// Mitsubishi GX Works2 project: 41715072   PLC: Q00J

PROGRAM MAIN
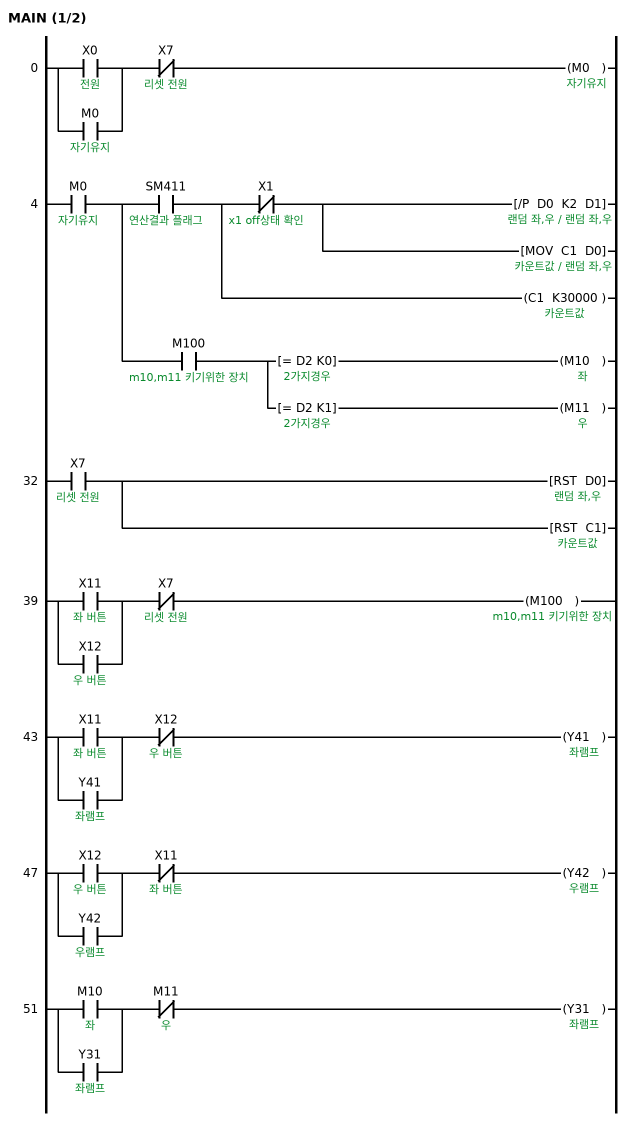
0     LD      X0  ; 전원
      OR      M0  ; 자기유지
      ANI     X7  ; 리셋 전원
      OUT     M0  ; 자기유지
4     LD      M0  ; 자기유지
      MPS
      AND     SM411  ; 연산결과 플래그
      MPS
      ANI     X1  ; x1 off상태 확인
      /P      D0 K2 D1  ; 랜덤 좌,우 / 랜덤 좌,우
      MOV     C1 D0  ; 카운트값
      MPP
      OUT     C1 K30000  ; 카운트값
      MPP
      AND     M100  ; m10,m11 키기위한 장치
      MPS
      AND=    D2 K0  ; 2가지경우
      OUT     M10  ; 좌
      MPP
      AND=    D2 K1  ; 2가지경우
      OUT     M11  ; 우
32    LD      X7  ; 리셋 전원
      RST     D0  ; 랜덤 좌,우
      RST     C1  ; 카운트값
39    LD      X11  ; 좌 버튼
      OR      X12  ; 우 버튼
      ANI     X7  ; 리셋 전원
      OUT     M100  ; m10,m11 키기위한 장치
43    LD      X11  ; 좌 버튼
      OR      Y41  ; 좌램프
      ANI     X12  ; 우 버튼
      OUT     Y41  ; 좌램프
47    LD      X12  ; 우 버튼
      OR      Y42  ; 우램프
      ANI     X11  ; 좌 버튼
      OUT     Y42  ; 우램프
51    LD      M10  ; 좌
      OR      Y31  ; 좌램프
      ANI     M11  ; 우
      OUT     Y31  ; 좌램프
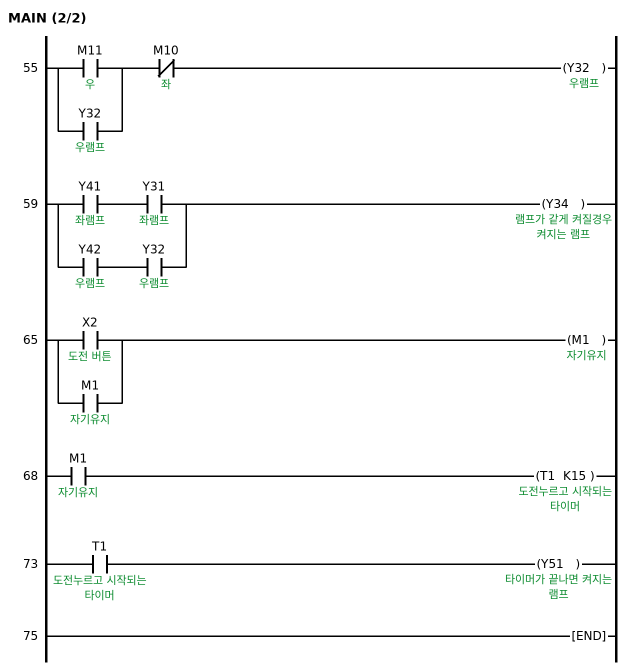
55    LD      M11  ; 우
      OR      Y32  ; 우램프
      ANI     M10  ; 좌
      OUT     Y32  ; 우램프
59    LD      Y41  ; 좌램프
      AND     Y31  ; 좌램프
      LD      Y42  ; 우램프
      AND     Y32  ; 우램프
      ORB
      OUT     Y34  ; 램프가 같게 켜질경우 켜지는 램프
65    LD      X2  ; 도전 버튼
      OR      M1  ; 자기유지
      OUT     M1  ; 자기유지
68    LD      M1  ; 자기유지
      OUT     T1 K15  ; 도전누르고 시작되는 타이머
73    LD      T1  ; 도전누르고 시작되는 타이머
      OUT     Y51  ; 타이머가 끝나면 켜지는 램프
75    END
END_PROGRAM
